{attribute addProperty BoxType "EL9227-4433-0018"}
{attribute addProperty Id "OCP_Inputs_ChannelAT %I*ARRAY[0..1] OF OCP_Inputs_Channel_8753EDC6192240OCP_Outputs_ChannelAT %Q*ARRAY[0..1] OF OCP_Outputs_Channel_F330A9163240WcStateAT %I*WcState_F855686C1620InfoDataAT %I*InfoData_BC63D37F80100"}
{attribute addProperty CRC "509652692"}
{attribute addProperty SizeInBites "320"}
{attribute addProperty SizeInBytes "40"}
TYPE EL9227_9EBC8997 :
STRUCT
	{attribute addProperty Name "OCP_Inputs_Channel"}
	OCP_Inputs_Channel : ARRAY[0..1] OF OCP_Inputs_Channel_8753EDC6;
	{attribute addProperty Name "OCP_Outputs_Channel"}
	OCP_Outputs_Channel : ARRAY[0..1] OF OCP_Outputs_Channel_F330A916;
	{attribute addProperty Name "WcState"}
	WcState : WcState_F855686C;
	{attribute addProperty Name "InfoData"}
	InfoData : InfoData_BC63D37F;
END_STRUCT
END_TYPE

(* stored: Version 1.2.0.0, ProductVersion 3.1.4024.9
   DUT EL9227_9EBC8997: Id {743502e1-f5ba-4670-9a25-b7825628777e} *)
